TYPE ST_LinearMotors :
STRUCT
	ID_Linear		: INT;
	pump1			: STRING(100);
	pump2			: STRING(100);
	pump3			: STRING(100);
	pump4			: STRING(100);
	pump5			: STRING(100);
	pump6			: STRING(100);
	pump7			: STRING(100);
	pump8			: STRING(100);
	pump9			: STRING(100);
	pump10			: STRING(100);
END_STRUCT
END_TYPE

(* stored: Version 1.1.0.1, ProductVersion 3.1.4024.15
   DUT ST_LinearMotors: Id {2f48993c-822d-4c5a-8367-a2c542e63700} *)
